INTERFACE ITF_ControlElement1 EXTENDS ITF_BaseControlElement

END_INTERFACE

(* stored: Version 1.1.0.1, ProductVersion 3.1.4024.15
   Itf ITF_ControlElement1: Id {147d77bc-fbf7-443b-894e-104deb3e854e} *)
